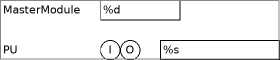
VISUALIZATION _VISU_ModuleMaster  // 280x60
VAR_IN_OUT
	mInst : FB_ModuleMaster;
END_VAR
    Rectangle (160,40 120x20), "%s", tooltip "%s", text variable: mInst._pPU^._activeJob^._sActiveJobDef.sJobSettings.aI_JobName, colour toggle: mInst._pPU^._activeJob <> 0
        p4168582468: mInst._pPU^._activeJob^._sActiveJobDef.sJobSettings.aI_JobName
    Ellipse (100,40 20x20), "I", colour toggle: mInst._pPU^._pAdsPu^.sI_Start.bI_Command OR mInst._pPU^._pAdsPu^.sI_Start.bO_CommandCanEx
        tap mInst._pPU^._pAdsPu^.sI_Start.bI_Command
    Ellipse (120,40 20x20), "O", colour toggle: mInst._pPU^._pAdsPu^.sI_Stop.bI_Command OR mInst._pPU^._pAdsPu^.sI_Stop.bO_CommandCanEx
        tap mInst._pPU^._pAdsPu^.sI_Stop.bI_Command
    Rectangle (100,0 80x20), "%d", tooltip "Master module idx", text variable: mInst._pMasterModule^._nIdx
    Rectangle (0,0 100x20), "MasterModule"
    Rectangle (0,40 100x20), "PU"
END_VISUALIZATION

(* stored: Version 1.1.0.1, ProductVersion 3.1.4024.11
   Visu _VISU_ModuleMaster: Id {c1d8c7a3-7d0d-4a3b-9a26-2906f1530475} *)
